// TIA Portal V18 export
TYPE "MEStoPLC_MainCheckOut_ext"
// stored: IsFailsafeCompliant false
   STRUCT
      UnloadLoad_ResultsStored1OK : Bool;   // UnUnloadLoading part process - Results stored OK
      UnloadLoad_ResultsStored1NG : Bool;   // UnUnloadLoading part process - Results stored NG
      UnloadLoad_ResultsStored1ReqMesDone : Bool;   // 存储完成，PLC复位 Station*DataSaveReq
      UnloadLoad_ResultsStored1Spare : Bool;   // Spare
      UnloadLoad_ResultsStored1Spare1 : Bool;   // Spare
      UnloadLoad_ResultsStored1Spare2 : Bool;   // Spare
      UnloadLoad_ResultsStored1Spare3 : Bool;   // Spare
      UnloadLoad_ResultsStored1Spare4 : Bool;   // Spare
      UnloadLoad_ResultsStored2OK : Bool;   // UnUnloadLoading part process - Results stored OK
      UnloadLoad_ResultsStored2NG : Bool;   // UnUnloadLoading part process - Results stored NG
      UnloadLoad_ResultsStored2ReqMesDone : Bool;   // 存储完成，PLC复位 Station*DataSaveReq
      UnloadLoad_ResultsStored2Spare : Bool;   // Spare
      UnloadLoad_ResultsStored2Spare1 : Bool;   // Spare
      UnloadLoad_ResultsStored2Spare2 : Bool;   // Spare
      UnloadLoad_ResultsStored2Spare3 : Bool;   // Spare
      UnloadLoad_ResultsStored2Spare4 : Bool;   // Spare
      UnloadLoad_ResultsStored3OK : Bool;   // 订单号
      UnloadLoad_ResultsStored3NG : Bool;   // UnUnloadLoading part process - Results stored OK
      UnloadLoad_ResultsStored3ReqMesDone : Bool;   // UnUnloadLoading part process - Results stored NG
      UnloadLoad_ResultsStored3Spare : Bool;   // 存储完成，PLC复位 Station*DataSaveReq
      UnloadLoad_ResultsStored3Spare1 : Bool;   // Spare
      UnloadLoad_ResultsStored3Spare2 : Bool;   // Spare
      UnloadLoad_ResultsStored3Spare3 : Bool;   // Spare
      UnloadLoad_ResultsStored3Spare4 : Bool;   // Spare
      UnloadLoad_ResultsStored4OK : Bool;   // UnUnloadLoading part process - Results stored OK
      UnloadLoad_ResultsStored4NG : Bool;   // UnUnloadLoading part process - Results stored NG
      UnloadLoad_ResultsStored4ReqMesDone : Bool;   // 存储完成，PLC复位 Station*DataSaveReq
      UnloadLoad_ResultsStored4Spare : Bool;   // Spare
      UnloadLoad_ResultsStored4Spare1 : Bool;   // Spare
      UnloadLoad_ResultsStored4Spare2 : Bool;   // Spare
      UnloadLoad_ResultsStored4Spare3 : Bool;   // Spare
      UnloadLoad_ResultsStored4Spare4 : Bool;   // Spare
      UnloadLoad_ResultsStored5OK : Bool;   // UnUnloadLoading part process - Results stored OK
      UnloadLoad_ResultsStored5NG : Bool;   // UnUnloadLoading part process - Results stored NG
      UnloadLoad_ResultsStored5ReqMesDone : Bool;   // 存储完成，PLC复位 Station*DataSaveReq
      UnloadLoad_ResultsStored5Spare : Bool;   // Spare
      UnloadLoad_ResultsStored5Spare1 : Bool;   // Spare
      UnloadLoad_ResultsStored5Spare2 : Bool;   // Spare
      UnloadLoad_ResultsStored5Spare3 : Bool;   // Spare
      UnloadLoad_ResultsStored5Spare4 : Bool;   // Spare
      UnloadLoad_ResultsStored6OK : Bool;   // UnUnloadLoading part process - Results stored OK
      UnloadLoad_ResultsStored6NG : Bool;   // UnUnloadLoading part process - Results stored NG
      UnloadLoad_ResultsStored6ReqMesDone : Bool;   // 存储完成，PLC复位 Station*DataSaveReq
      UnloadLoad_ResultsStored6Spare : Bool;   // Spare
      UnloadLoad_ResultsStored6Spare1 : Bool;   // Spare
      UnloadLoad_ResultsStored6Spare2 : Bool;   // Spare
      UnloadLoad_ResultsStored6Spare3 : Bool;   // Spare
      UnloadLoad_ResultsStored6Spare4 : Bool;   // Spare
      UnloadLoad_ResultsStored7OK : Bool;   // UnUnloadLoading part process - Results stored OK
      UnloadLoad_ResultsStored7NG : Bool;   // UnUnloadLoading part process - Results stored NG
      UnloadLoad_ResultsStored7ReqMesDone : Bool;   // 存储完成，PLC复位 Station*DataSaveReq
      UnloadLoad_ResultsStored7Spare : Bool;   // Spare
      UnloadLoad_ResultsStored7Spare1 : Bool;   // Spare
      UnloadLoad_ResultsStored7Spare2 : Bool;   // Spare
      UnloadLoad_ResultsStored7Spare3 : Bool;   // Spare
      UnloadLoad_ResultsStored7Spare4 : Bool;   // Spare
      UnloadLoad_ResultsStored8OK : Bool;   // UnUnloadLoading part process - Results stored OK
      UnloadLoad_ResultsStored8NG : Bool;   // UnUnloadLoading part process - Results stored NG
      UnloadLoad_ResultsStored8ReqMesDone : Bool;   // 存储完成，PLC复位 Station*DataSaveReq
      UnloadLoad_ResultsStored8Spare : Bool;   // Spare
      UnloadLoad_ResultsStored8Spare5 : Bool;   // Spare
      UnloadLoad_ResultsStored8Spare6 : Bool;   // Spare
      UnloadLoad_ResultsStored8Spare8 : Bool;   // Spare
      UnloadLoad_ResultsStored8Spare9 : Bool;   // Spare
   END_STRUCT;
END_TYPE
